(* CODESYS project waterTankFunctionsAndBlocks.export

Project tree, tasks and I/O mapping:
  Device : CODESYS Control Win V3 x64, CODESYS, version 3.5.22.30
    application Application
      libraries: Standard, 3.5.22.0 (System)
      task MainTask (cyclic, interval t#20ms, priority 1) calls PLC_PRG
      function FC_Scaling [LD]
      program PLC_PRG [LD]
      Symbols
*)

// Device/Application/PLC_PRG
PROGRAM PLC_PRG
VAR
	Pot1_Fill: REAL;
	Tank1_Fill: REAL;
	Pot2_Discharge: REAL;
	Tank1_DischargeValve: REAL;
	Error1: BOOL;
	Tank1_LevelMeter: REAL;
	WaterLevel: REAL;
	Error2: BOOL;
	Display1_WaterLevel: INT;
	Tank1_FlowMeter: REAL;
	FlowMeter: REAL;
	Error3: BOOL;
	
	Display2_FlowRate: INT;
END_VAR

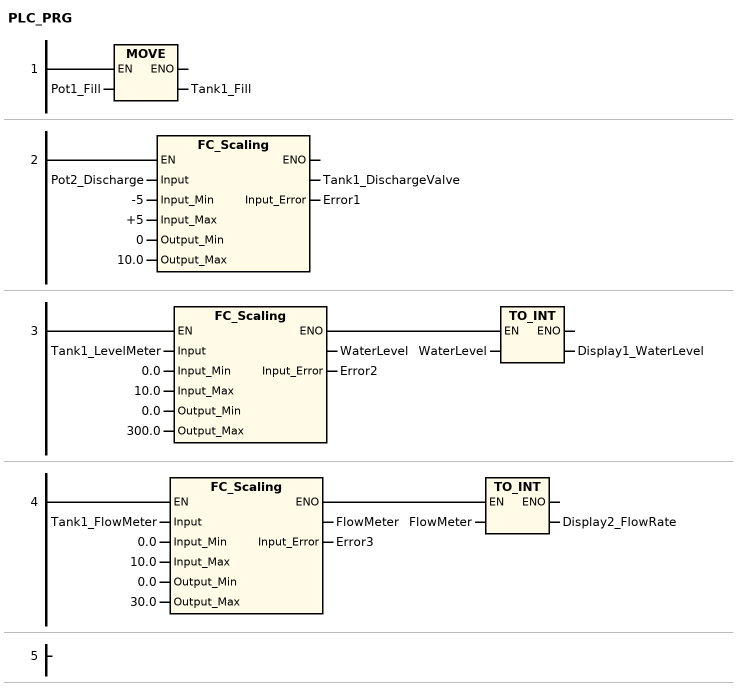
// NETWORK 1
Tank1_Fill := Pot1_Fill;

// NETWORK 2
Tank1_DischargeValve := FC_Scaling(Input := Pot2_Discharge, Input_Min := -5, Input_Max := +5, Output_Min := 0, Output_Max := 10.0, Input_Error => Error1);

// NETWORK 3
WaterLevel := FC_Scaling(Input := Tank1_LevelMeter, Input_Min := 0.0, Input_Max := 10.0, Output_Min := 0.0, Output_Max := 300.0, Input_Error => Error2);
Display1_WaterLevel := TO_INT(WaterLevel);

// NETWORK 4
FlowMeter := FC_Scaling(Input := Tank1_FlowMeter, Input_Min := 0.0, Input_Max := 10.0, Output_Min := 0.0, Output_Max := 30.0, Input_Error => Error3);
Display2_FlowRate := TO_INT(FlowMeter);

// NETWORK 5

END_PROGRAM

// Device/Application/FC_Scaling
FUNCTION FC_Scaling : REAL
VAR_INPUT
	Input: REAL;
	Input_Min: REAL;
	Input_Max: REAL;
	Output_Min: REAL;
	Output_Max: REAL;
END_VAR
VAR
	Var1: REAL;
	Var2: REAL;
	Var3: REAL;
	Var4: REAL;
	Var5: REAL;
END_VAR

VAR_OUTPUT
	Input_Error: BOOL;
END_VAR

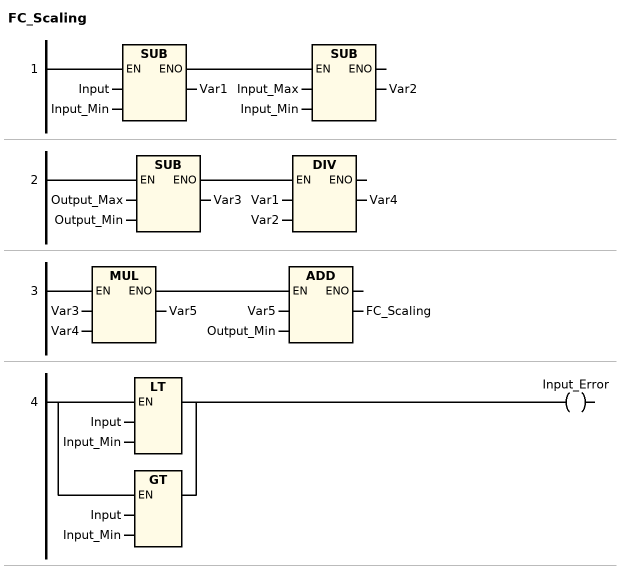
// NETWORK 1
Var1 := Input - Input_Min;
Var2 := Input_Max - Input_Min;

// NETWORK 2
Var3 := Output_Max - Output_Min;
Var4 := Var1 / Var2;

// NETWORK 3
Var5 := Var3 * Var4;
FC_Scaling := Var5 + Output_Min;

// NETWORK 4
Input_Error := Input < Input_Min OR Input > Input_Min;

END_FUNCTION
